(* Logix 5000 project; controller L3 vendor 1 type 14 code 92 rev 20.12; software revision 20.04; part 5 of 9 *)
(* tags used below, declared in another part *)
   B3 : DINT[100];
   cligno : BOOL;
   Status : INT;   // INT tag to retrieve Status value through GSV created during conversion
   T4 : TIMER[180];
   t_minute : TIMER;   // tempo on toutes les minute
   t_seconde : TIMER;   // tempo on toutes les secondes
   tcligno : TIMER;
(* _2_GENERAL, continued *)

ROUTINE _2_GENERAL   (* ladder *)
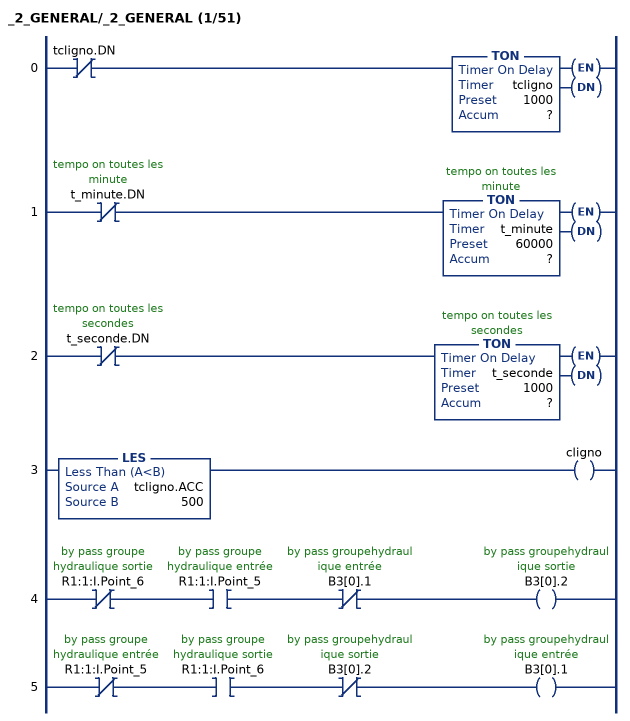
   0: XIO(tcligno.DN)TON(tcligno,?,?);
   1: XIO(t_minute.DN)TON(t_minute,?,?);
   2: XIO(t_seconde.DN)TON(t_seconde,?,?);
   3: LES(tcligno.ACC,500)OTE(cligno);
   4: XIO(R1:1:I.Point_6)XIC(R1:1:I.Point_5)XIO(B3[0].1)OTE(B3[0].2);
   5: XIO(R1:1:I.Point_5)XIC(R1:1:I.Point_6)XIO(B3[0].2)OTE(B3[0].1);
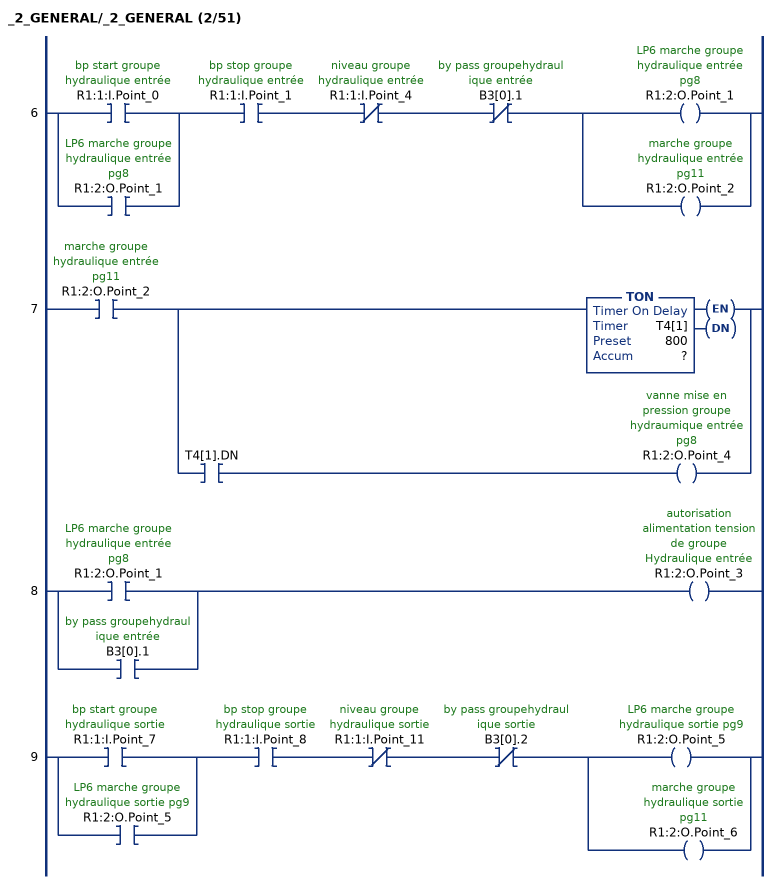
   6: [XIC(R1:1:I.Point_0) ,XIC(R1:2:O.Point_1) ]XIC(R1:1:I.Point_1)XIO(R1:1:I.Point_4)XIO(B3[0].1)[OTE(R1:2:O.Point_1) ,OTE(R1:2:O.Point_2) ];
   7: XIC(R1:2:O.Point_2)[TON(T4[1],?,?) ,XIC(T4[1].DN) OTE(R1:2:O.Point_4) ];
   8: [XIC(R1:2:O.Point_1) ,XIC(B3[0].1) ]OTE(R1:2:O.Point_3);
   9: [XIC(R1:1:I.Point_7) ,XIC(R1:2:O.Point_5) ]XIC(R1:1:I.Point_8)XIO(R1:1:I.Point_11)XIO(B3[0].2)[OTE(R1:2:O.Point_5) ,OTE(R1:2:O.Point_6) ];
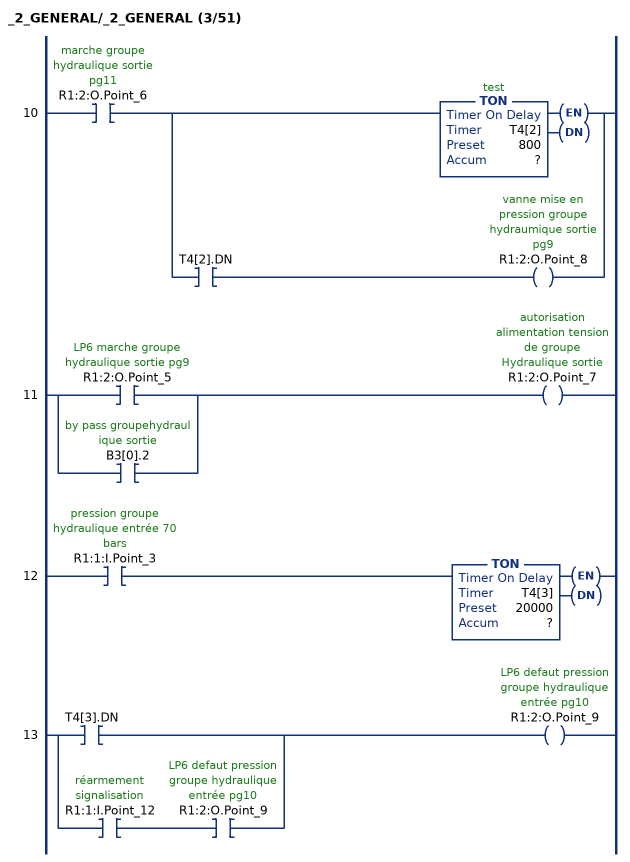
   10: XIC(R1:2:O.Point_6)[TON(T4[2],?,?) ,XIC(T4[2].DN) OTE(R1:2:O.Point_8) ];
   11: [XIC(R1:2:O.Point_5) ,XIC(B3[0].2) ]OTE(R1:2:O.Point_7);
   12: XIC(R1:1:I.Point_3)TON(T4[3],?,?);
   13: [XIC(T4[3].DN) ,XIC(R1:1:I.Point_12) XIC(R1:2:O.Point_9) ]OTE(R1:2:O.Point_9);
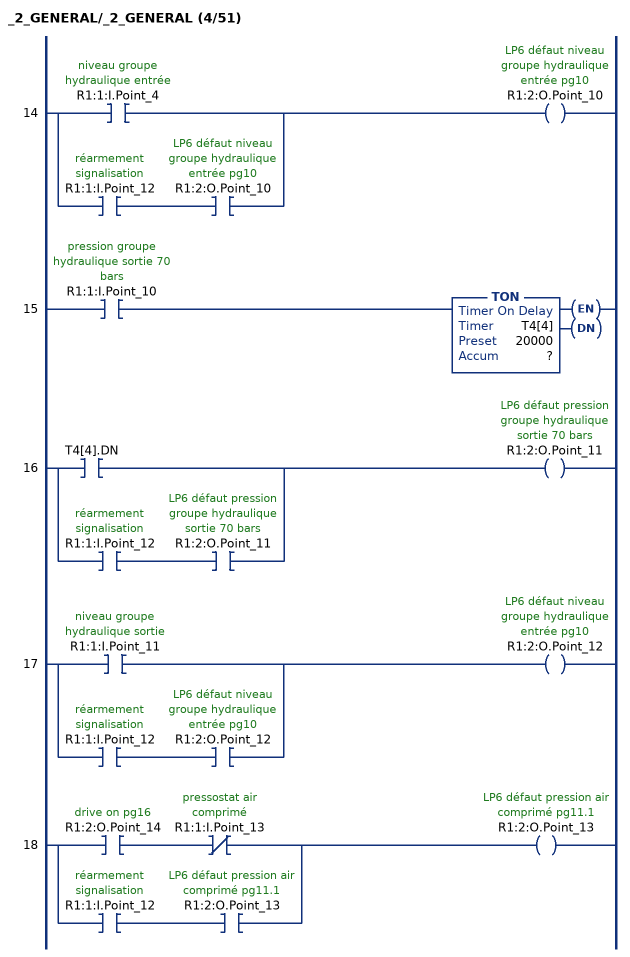
   14: [XIC(R1:1:I.Point_4) ,XIC(R1:1:I.Point_12) XIC(R1:2:O.Point_10) ]OTE(R1:2:O.Point_10);
   15: XIC(R1:1:I.Point_10)TON(T4[4],?,?);
   16: [XIC(T4[4].DN) ,XIC(R1:1:I.Point_12) XIC(R1:2:O.Point_11) ]OTE(R1:2:O.Point_11);
   17: [XIC(R1:1:I.Point_11) ,XIC(R1:1:I.Point_12) XIC(R1:2:O.Point_12) ]OTE(R1:2:O.Point_12);
   18: [XIC(R1:2:O.Point_14) XIO(R1:1:I.Point_13) ,XIC(R1:1:I.Point_12) XIC(R1:2:O.Point_13) ]OTE(R1:2:O.Point_13);
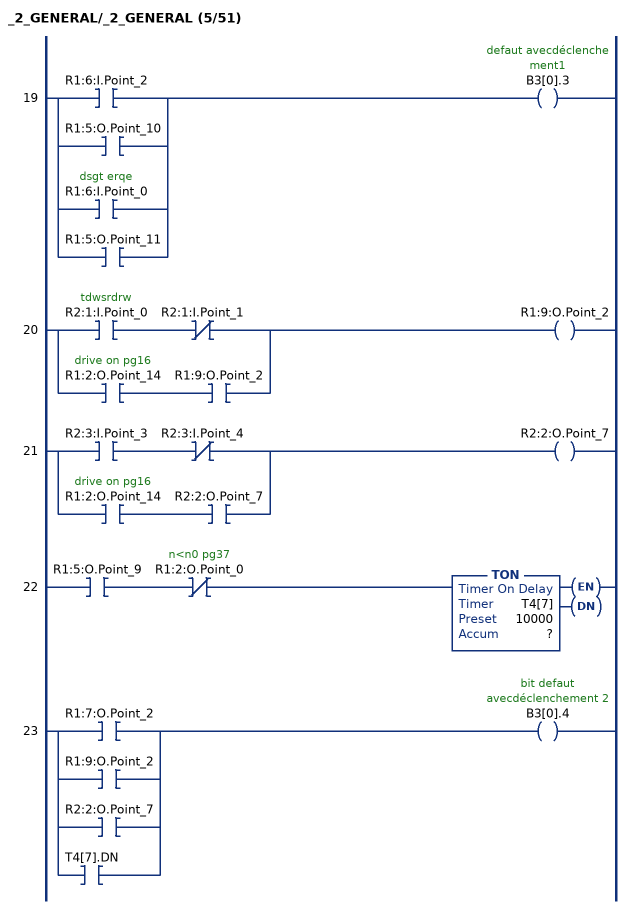
   19: [XIC(R1:6:I.Point_2) ,XIC(R1:5:O.Point_10) ,XIC(R1:6:I.Point_0) ,XIC(R1:5:O.Point_11) ]OTE(B3[0].3);
   20: [XIC(R2:1:I.Point_0) XIO(R2:1:I.Point_1) ,XIC(R1:2:O.Point_14) XIC(R1:9:O.Point_2) ]OTE(R1:9:O.Point_2);
   21: [XIC(R2:3:I.Point_3) XIO(R2:3:I.Point_4) ,XIC(R1:2:O.Point_14) XIC(R2:2:O.Point_7) ]OTE(R2:2:O.Point_7);
   22: XIC(R1:5:O.Point_9)XIO(R1:2:O.Point_0)TON(T4[7],?,?);
   23: [XIC(R1:7:O.Point_2) ,XIC(R1:9:O.Point_2) ,XIC(R2:2:O.Point_7) ,XIC(T4[7].DN) ]OTE(B3[0].4);
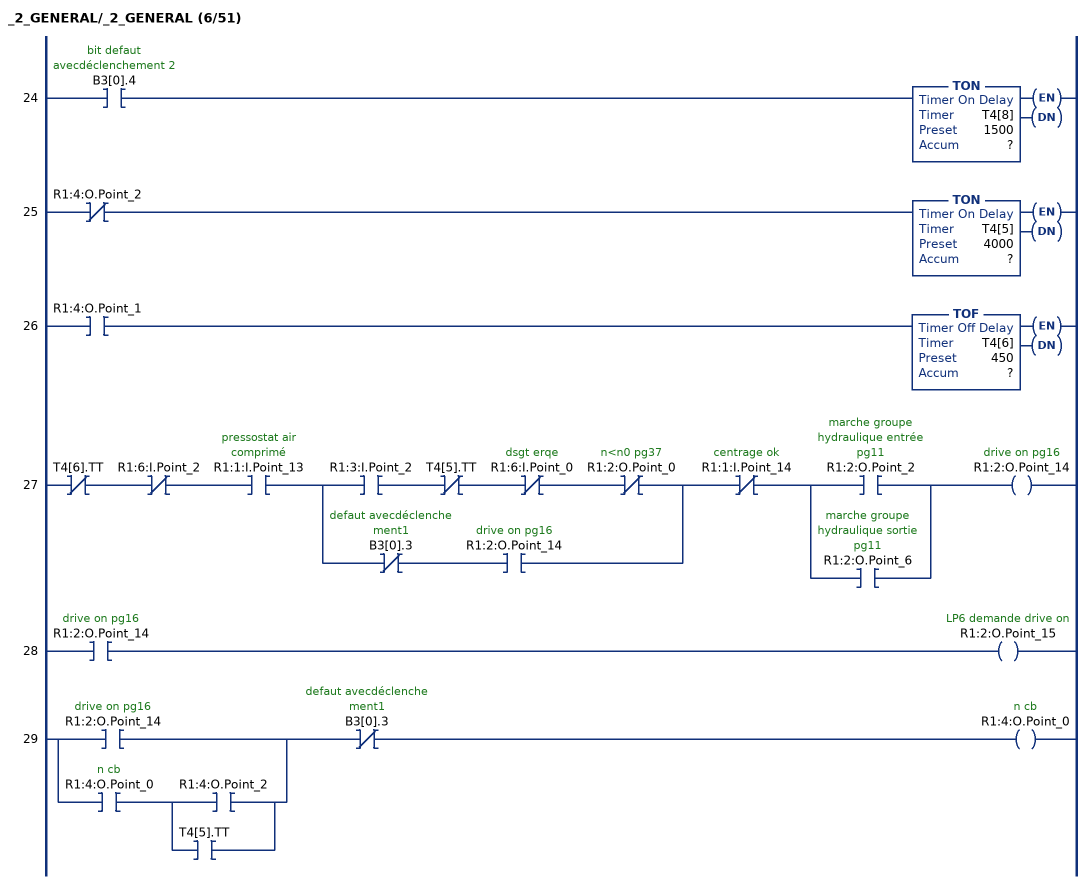
   24: XIC(B3[0].4)TON(T4[8],?,?);
   25: XIO(R1:4:O.Point_2)TON(T4[5],?,?);
   26: XIC(R1:4:O.Point_1)TOF(T4[6],?,?);
   27: XIO(T4[6].TT)XIO(R1:6:I.Point_2)XIC(R1:1:I.Point_13)[XIC(R1:3:I.Point_2) XIO(T4[5].TT) XIO(R1:6:I.Point_0) XIO(R1:2:O.Point_0) ,XIO(B3[0].3) XIC(R1:2:O.Point_14) ]XIO(R1:1:I.Point_14)[XIC(R1:2:O.Point_2) ,XIC(R1:2:O.Point_6) ]OTE(R1:2:O.Point_14);
   28: XIC(R1:2:O.Point_14)OTE(R1:2:O.Point_15);
   29: [XIC(R1:2:O.Point_14) ,XIC(R1:4:O.Point_0) [XIC(R1:4:O.Point_2) ,XIC(T4[5].TT) ] ]XIO(B3[0].3)OTE(R1:4:O.Point_0);
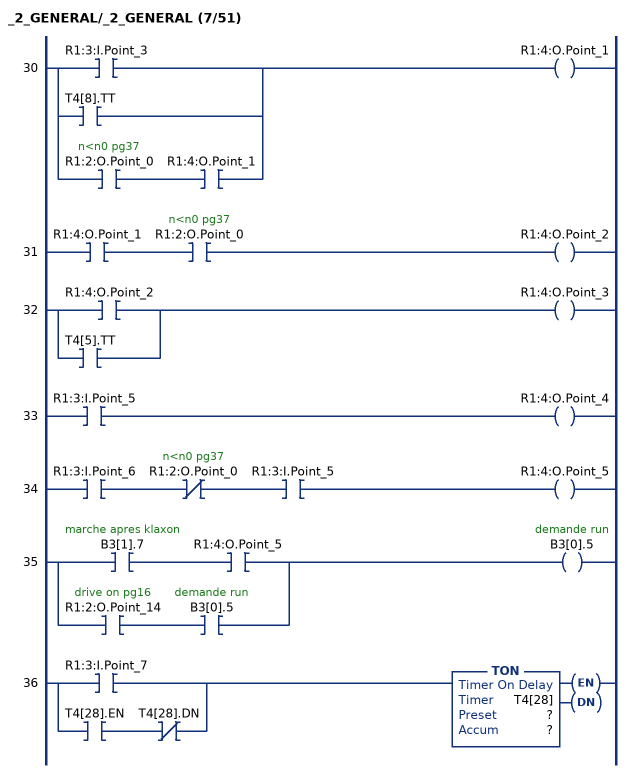
   30: [XIC(R1:3:I.Point_3) ,XIC(T4[8].TT) ,XIC(R1:2:O.Point_0) XIC(R1:4:O.Point_1) ]OTE(R1:4:O.Point_1);
   31: XIC(R1:4:O.Point_1)XIC(R1:2:O.Point_0)OTE(R1:4:O.Point_2);
   32: [XIC(R1:4:O.Point_2) ,XIC(T4[5].TT) ]OTE(R1:4:O.Point_3);
   33: XIC(R1:3:I.Point_5)OTE(R1:4:O.Point_4);
   34: XIC(R1:3:I.Point_6)XIO(R1:2:O.Point_0)XIC(R1:3:I.Point_5)OTE(R1:4:O.Point_5);
   35: [XIC(B3[1].7) XIC(R1:4:O.Point_5) ,XIC(R1:2:O.Point_14) XIC(B3[0].5) ]OTE(B3[0].5);
   36: [XIC(R1:3:I.Point_7) ,XIC(T4[28].EN) XIO(T4[28].DN) ]TON(T4[28],?,?);
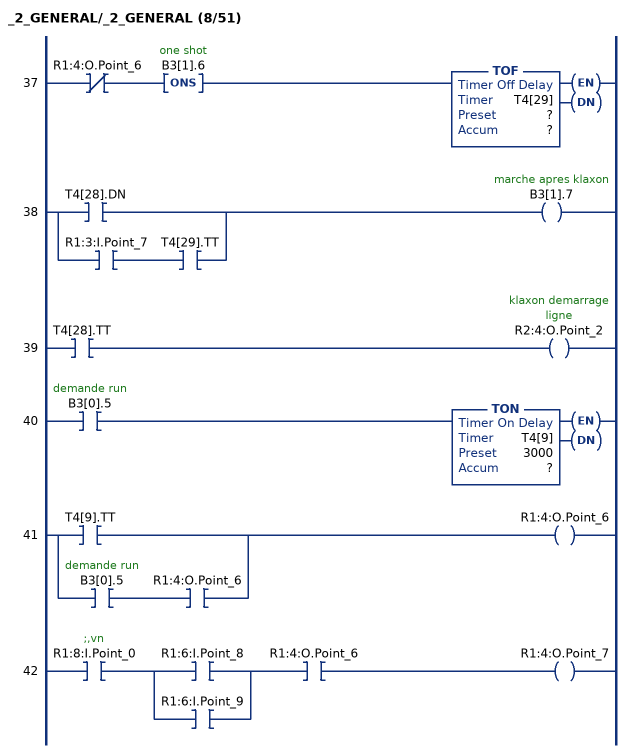
   37: XIO(R1:4:O.Point_6)ONS(B3[1].6)TOF(T4[29],?,?);
   38: [XIC(T4[28].DN) ,XIC(R1:3:I.Point_7) XIC(T4[29].TT) ]OTE(B3[1].7);
   39: XIC(T4[28].TT)OTE(R2:4:O.Point_2);
   40: XIC(B3[0].5)TON(T4[9],?,?);
   41: [XIC(T4[9].TT) ,XIC(B3[0].5) XIC(R1:4:O.Point_6) ]OTE(R1:4:O.Point_6);
   42: XIC(R1:8:I.Point_0)[XIC(R1:6:I.Point_8) ,XIC(R1:6:I.Point_9) ]XIC(R1:4:O.Point_6)OTE(R1:4:O.Point_7);
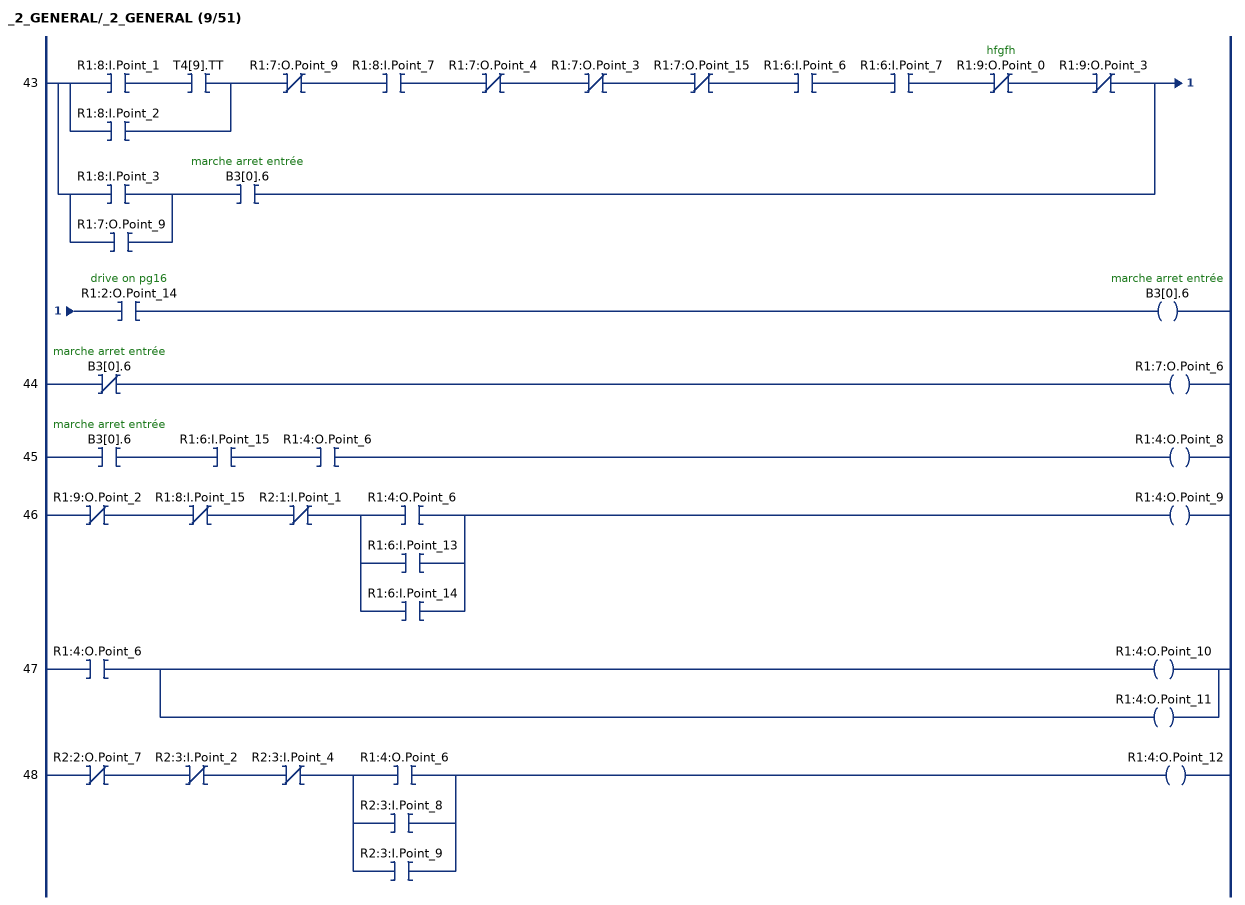
   43: [[XIC(R1:8:I.Point_1) XIC(T4[9].TT) ,XIC(R1:8:I.Point_2) ] XIO(R1:7:O.Point_9) XIC(R1:8:I.Point_7) XIO(R1:7:O.Point_4) XIO(R1:7:O.Point_3) XIO(R1:7:O.Point_15) XIC(R1:6:I.Point_6) XIC(R1:6:I.Point_7) XIO(R1:9:O.Point_0) XIO(R1:9:O.Point_3) ,[XIC(R1:8:I.Point_3) ,XIC(R1:7:O.Point_9) ] XIC(B3[0].6) ]XIC(R1:2:O.Point_14)OTE(B3[0].6);
   44: XIO(B3[0].6)OTE(R1:7:O.Point_6);
   45: XIC(B3[0].6)XIC(R1:6:I.Point_15)XIC(R1:4:O.Point_6)OTE(R1:4:O.Point_8);
   46: XIO(R1:9:O.Point_2)XIO(R1:8:I.Point_15)XIO(R2:1:I.Point_1)[XIC(R1:4:O.Point_6) ,XIC(R1:6:I.Point_13) ,XIC(R1:6:I.Point_14) ]OTE(R1:4:O.Point_9);
   47: XIC(R1:4:O.Point_6)[OTE(R1:4:O.Point_10) ,OTE(R1:4:O.Point_11) ];
   48: XIO(R2:2:O.Point_7)XIO(R2:3:I.Point_2)XIO(R2:3:I.Point_4)[XIC(R1:4:O.Point_6) ,XIC(R2:3:I.Point_8) ,XIC(R2:3:I.Point_9) ]OTE(R1:4:O.Point_12);
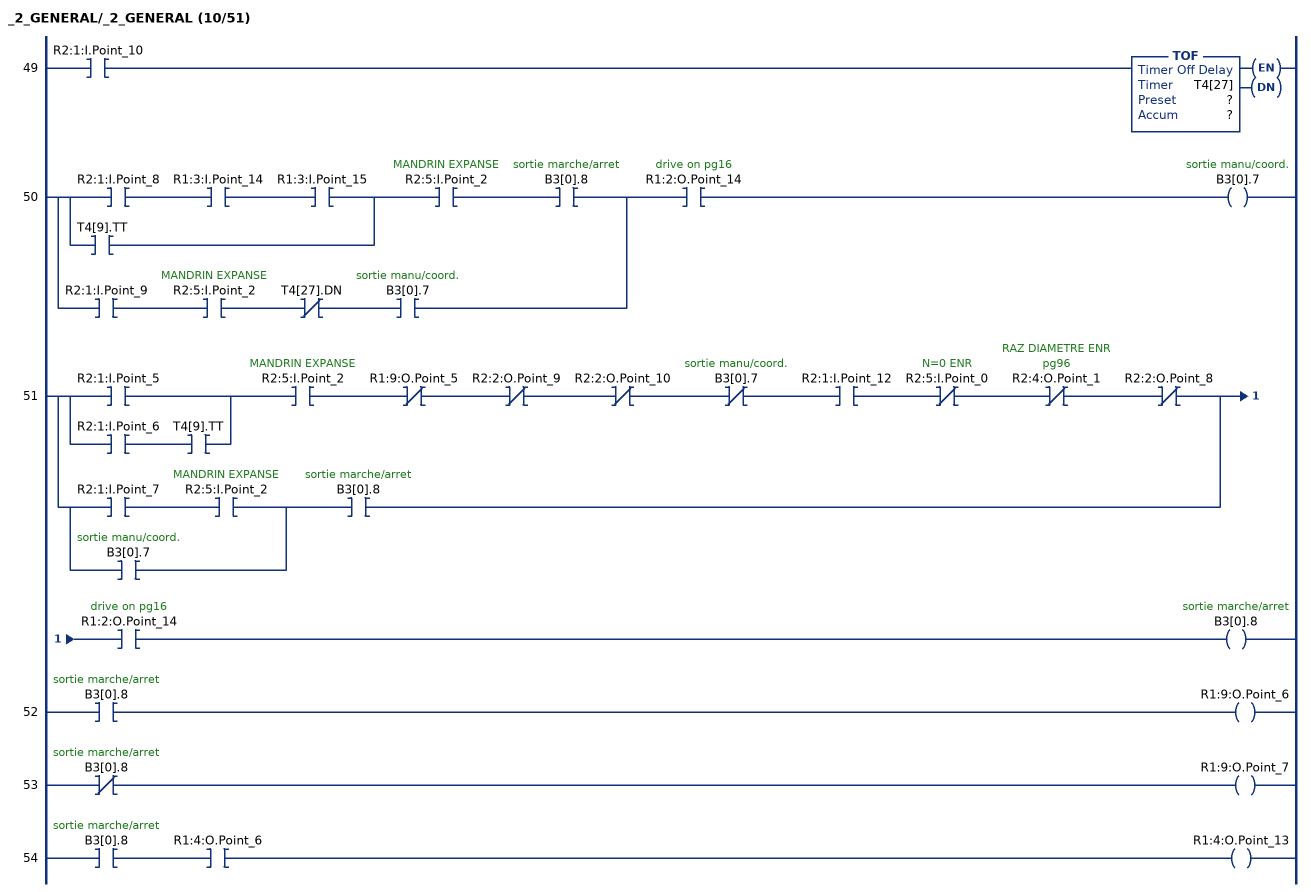
   49: XIC(R2:1:I.Point_10)TOF(T4[27],?,?);
   50: [[XIC(R2:1:I.Point_8) XIC(R1:3:I.Point_14) XIC(R1:3:I.Point_15) ,XIC(T4[9].TT) ] XIC(R2:5:I.Point_2) XIC(B3[0].8) ,XIC(R2:1:I.Point_9) XIC(R2:5:I.Point_2) XIO(T4[27].DN) XIC(B3[0].7) ]XIC(R1:2:O.Point_14)OTE(B3[0].7);
   51: [[XIC(R2:1:I.Point_5) ,XIC(R2:1:I.Point_6) XIC(T4[9].TT) ] XIC(R2:5:I.Point_2) XIO(R1:9:O.Point_5) XIO(R2:2:O.Point_9) XIO(R2:2:O.Point_10) XIO(B3[0].7) XIC(R2:1:I.Point_12) XIO(R2:5:I.Point_0) XIO(R2:4:O.Point_1) XIO(R2:2:O.Point_8) ,[XIC(R2:1:I.Point_7) XIC(R2:5:I.Point_2) ,XIC(B3[0].7) ] XIC(B3[0].8) ]XIC(R1:2:O.Point_14)OTE(B3[0].8);
   52: XIC(B3[0].8)OTE(R1:9:O.Point_6);
   53: XIO(B3[0].8)OTE(R1:9:O.Point_7);
   54: XIC(B3[0].8)XIC(R1:4:O.Point_6)OTE(R1:4:O.Point_13);
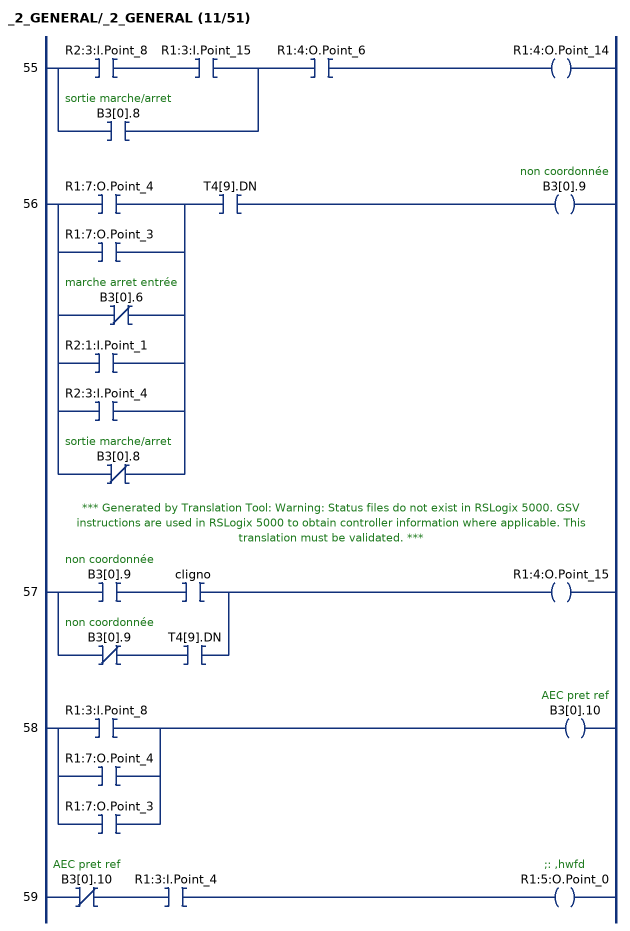
   55: [XIC(R2:3:I.Point_8) XIC(R1:3:I.Point_15) ,XIC(B3[0].8) ]XIC(R1:4:O.Point_6)OTE(R1:4:O.Point_14);
   56: [XIC(R1:7:O.Point_4) ,XIC(R1:7:O.Point_3) ,XIO(B3[0].6) ,XIC(R2:1:I.Point_1) ,XIC(R2:3:I.Point_4) ,XIO(B3[0].8) ]XIC(T4[9].DN)OTE(B3[0].9);
   // *** Generated by Translation Tool: Warning: Status files do not exist in RSLogix 5000. GSV instructions are used in RSLogix 5000 to obtain controller information where applicable. This translation must be validated. ***
   57: [XIC(B3[0].9) XIC(cligno) ,XIO(B3[0].9) XIC(T4[9].DN) ]OTE(R1:4:O.Point_15);
   58: [XIC(R1:3:I.Point_8) ,XIC(R1:7:O.Point_4) ,XIC(R1:7:O.Point_3) ]OTE(B3[0].10);
   59: XIO(B3[0].10)XIC(R1:3:I.Point_4)OTE(R1:5:O.Point_0);
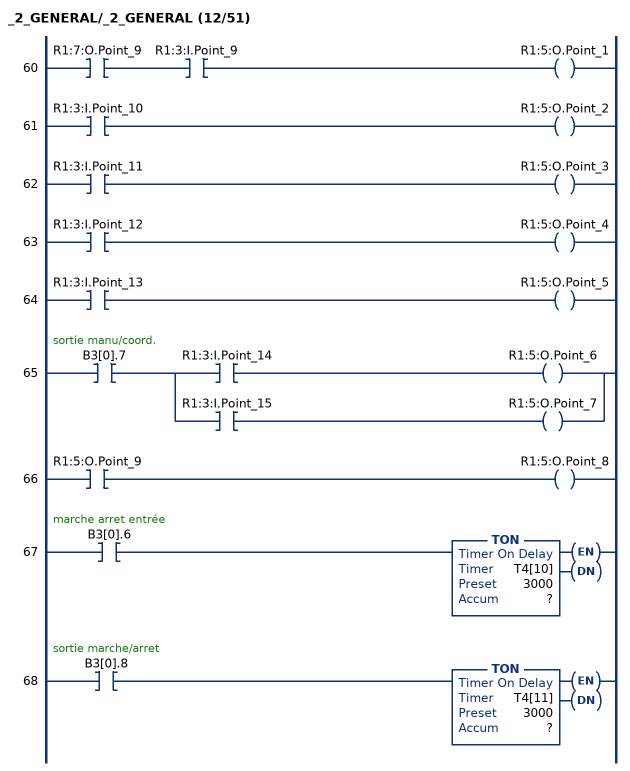
   60: XIC(R1:7:O.Point_9)XIC(R1:3:I.Point_9)OTE(R1:5:O.Point_1);
   61: XIC(R1:3:I.Point_10)OTE(R1:5:O.Point_2);
   62: XIC(R1:3:I.Point_11)OTE(R1:5:O.Point_3);
   63: XIC(R1:3:I.Point_12)OTE(R1:5:O.Point_4);
   64: XIC(R1:3:I.Point_13)OTE(R1:5:O.Point_5);
   65: XIC(B3[0].7)[XIC(R1:3:I.Point_14) OTE(R1:5:O.Point_6) ,XIC(R1:3:I.Point_15) OTE(R1:5:O.Point_7) ];
   66: XIC(R1:5:O.Point_9)OTE(R1:5:O.Point_8);
   67: XIC(B3[0].6)TON(T4[10],?,?);
   68: XIC(B3[0].8)TON(T4[11],?,?);
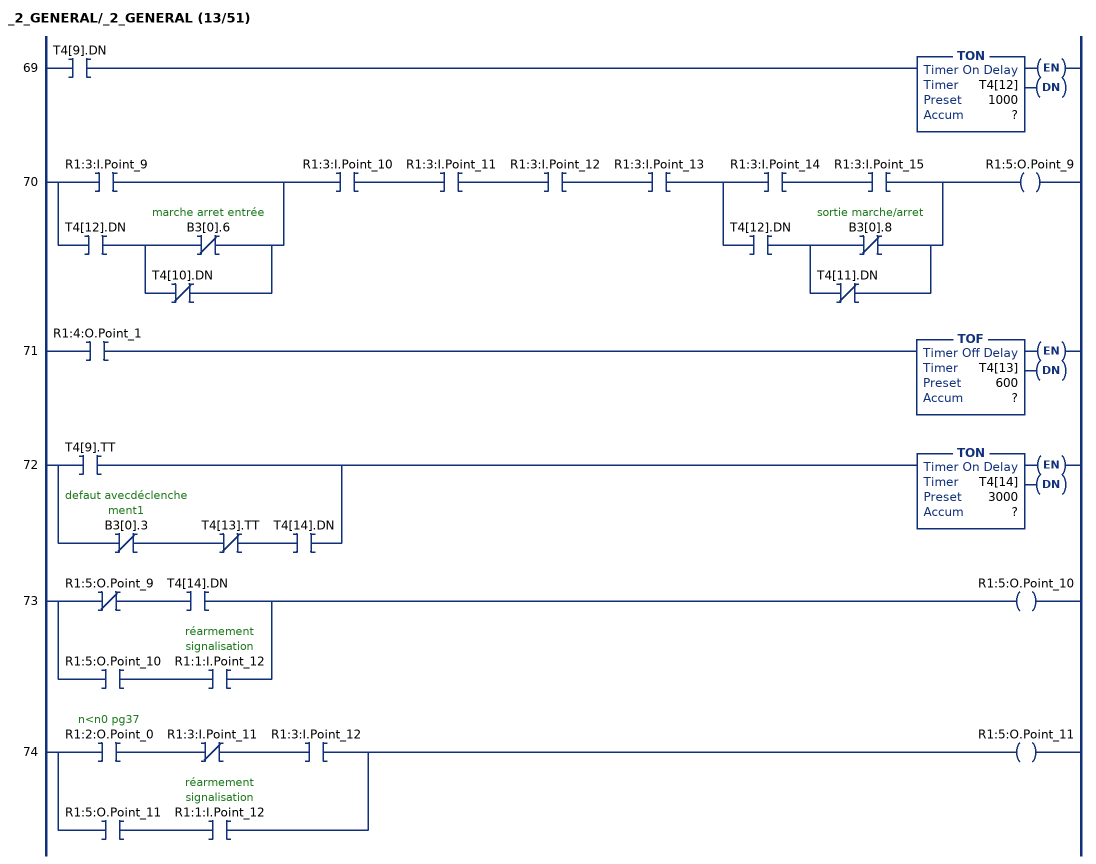
   69: XIC(T4[9].DN)TON(T4[12],?,?);
   70: [XIC(R1:3:I.Point_9) ,XIC(T4[12].DN) [XIO(B3[0].6) ,XIO(T4[10].DN) ] ]XIC(R1:3:I.Point_10)XIC(R1:3:I.Point_11)XIC(R1:3:I.Point_12)XIC(R1:3:I.Point_13)[XIC(R1:3:I.Point_14) XIC(R1:3:I.Point_15) ,XIC(T4[12].DN) [XIO(B3[0].8) ,XIO(T4[11].DN) ] ]OTE(R1:5:O.Point_9);
   71: XIC(R1:4:O.Point_1)TOF(T4[13],?,?);
   72: [XIC(T4[9].TT) ,XIO(B3[0].3) XIO(T4[13].TT) XIC(T4[14].DN) ]TON(T4[14],?,?);
   73: [XIO(R1:5:O.Point_9) XIC(T4[14].DN) ,XIC(R1:5:O.Point_10) XIC(R1:1:I.Point_12) ]OTE(R1:5:O.Point_10);
   74: [XIC(R1:2:O.Point_0) XIO(R1:3:I.Point_11) XIC(R1:3:I.Point_12) ,XIC(R1:5:O.Point_11) XIC(R1:1:I.Point_12) ]OTE(R1:5:O.Point_11);
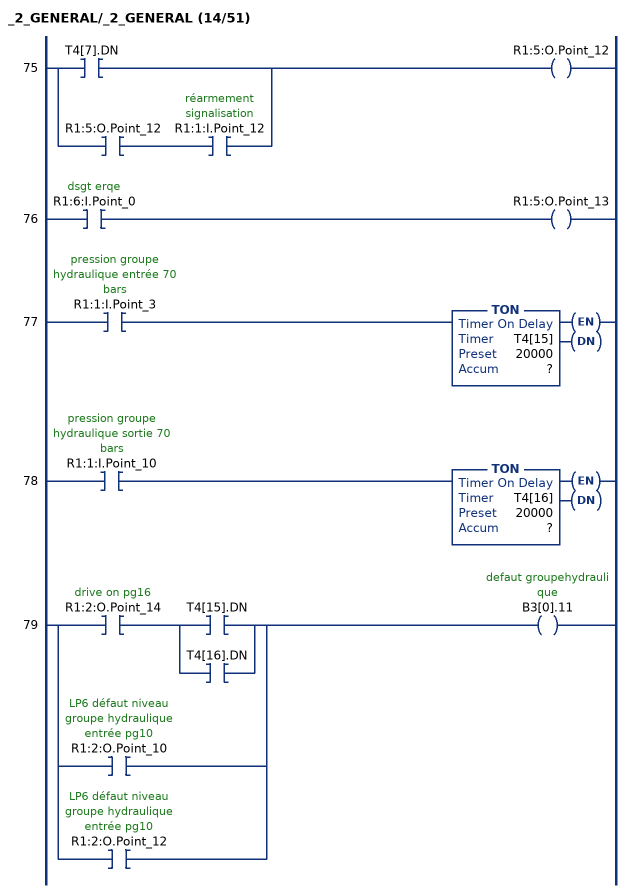
   75: [XIC(T4[7].DN) ,XIC(R1:5:O.Point_12) XIC(R1:1:I.Point_12) ]OTE(R1:5:O.Point_12);
   76: XIC(R1:6:I.Point_0)OTE(R1:5:O.Point_13);
   77: XIC(R1:1:I.Point_3)TON(T4[15],?,?);
   78: XIC(R1:1:I.Point_10)TON(T4[16],?,?);
   79: [XIC(R1:2:O.Point_14) [XIC(T4[15].DN) ,XIC(T4[16].DN) ] ,XIC(R1:2:O.Point_10) ,XIC(R1:2:O.Point_12) ]OTE(B3[0].11);
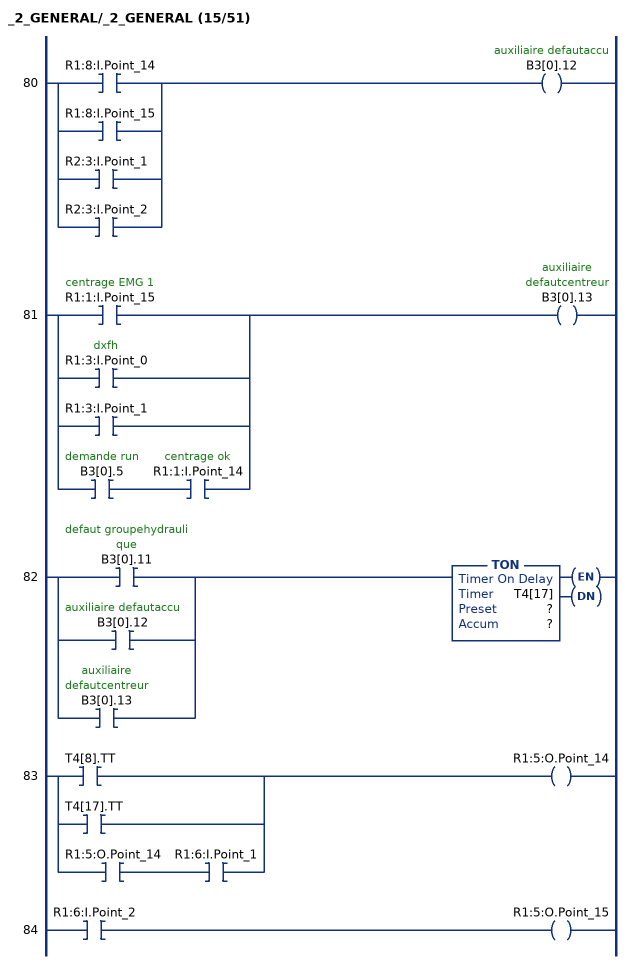
   80: [XIC(R1:8:I.Point_14) ,XIC(R1:8:I.Point_15) ,XIC(R2:3:I.Point_1) ,XIC(R2:3:I.Point_2) ]OTE(B3[0].12);
   81: [XIC(R1:1:I.Point_15) ,XIC(R1:3:I.Point_0) ,XIC(R1:3:I.Point_1) ,XIC(B3[0].5) XIC(R1:1:I.Point_14) ]OTE(B3[0].13);
   82: [XIC(B3[0].11) ,XIC(B3[0].12) ,XIC(B3[0].13) ]TON(T4[17],?,?);
   83: [XIC(T4[8].TT) ,XIC(T4[17].TT) ,XIC(R1:5:O.Point_14) XIC(R1:6:I.Point_1) ]OTE(R1:5:O.Point_14);
   84: XIC(R1:6:I.Point_2)OTE(R1:5:O.Point_15);
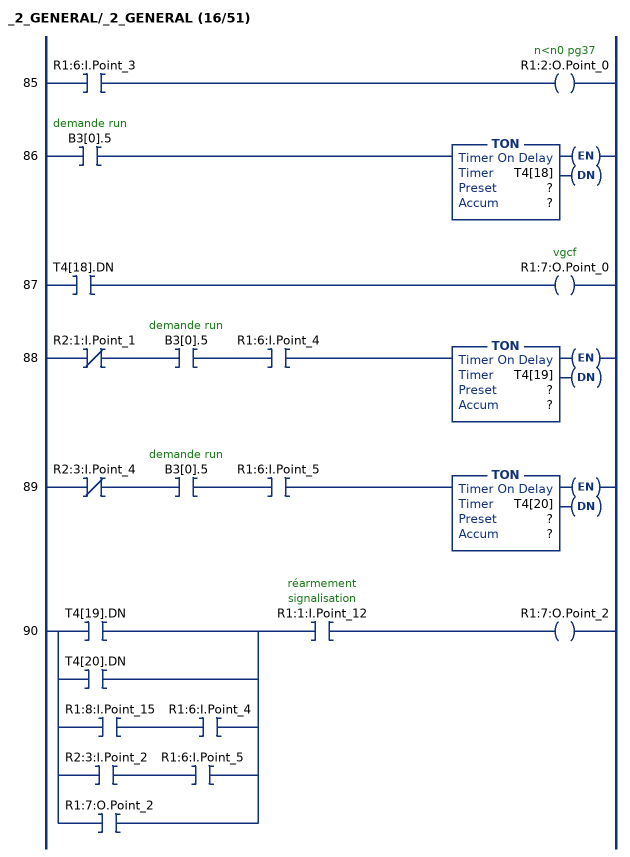
   85: XIC(R1:6:I.Point_3)OTE(R1:2:O.Point_0);
   86: XIC(B3[0].5)TON(T4[18],?,?);
   87: XIC(T4[18].DN)OTE(R1:7:O.Point_0);
   88: XIO(R2:1:I.Point_1)XIC(B3[0].5)XIC(R1:6:I.Point_4)TON(T4[19],?,?);
   89: XIO(R2:3:I.Point_4)XIC(B3[0].5)XIC(R1:6:I.Point_5)TON(T4[20],?,?);
   90: [XIC(T4[19].DN) ,XIC(T4[20].DN) ,XIC(R1:8:I.Point_15) XIC(R1:6:I.Point_4) ,XIC(R2:3:I.Point_2) XIC(R1:6:I.Point_5) ,XIC(R1:7:O.Point_2) ]XIC(R1:1:I.Point_12)OTE(R1:7:O.Point_2);
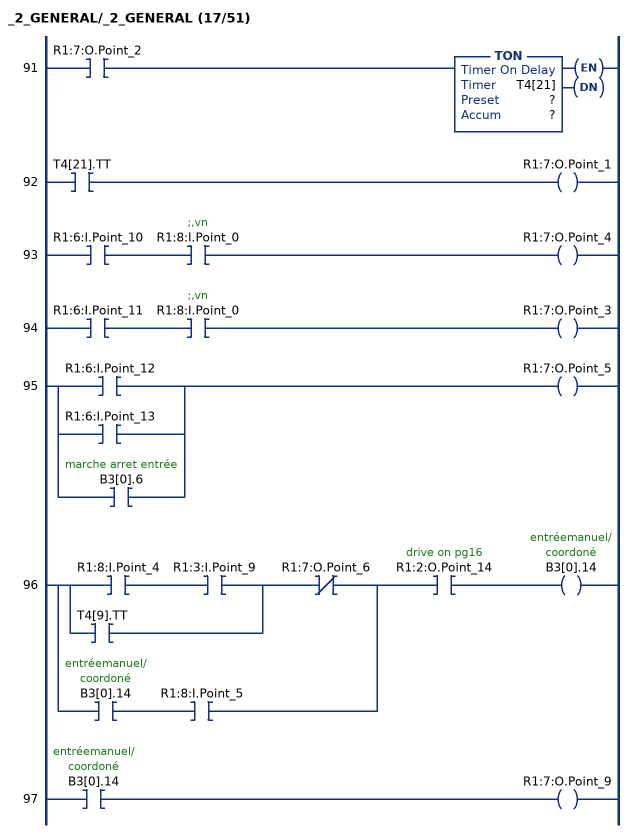
   91: XIC(R1:7:O.Point_2)TON(T4[21],?,?);
   92: XIC(T4[21].TT)OTE(R1:7:O.Point_1);
   93: XIC(R1:6:I.Point_10)XIC(R1:8:I.Point_0)OTE(R1:7:O.Point_4);
   94: XIC(R1:6:I.Point_11)XIC(R1:8:I.Point_0)OTE(R1:7:O.Point_3);
   95: [XIC(R1:6:I.Point_12) ,XIC(R1:6:I.Point_13) ,XIC(B3[0].6) ]OTE(R1:7:O.Point_5);
   96: [[XIC(R1:8:I.Point_4) XIC(R1:3:I.Point_9) ,XIC(T4[9].TT) ] XIO(R1:7:O.Point_6) ,XIC(B3[0].14) XIC(R1:8:I.Point_5) ]XIC(R1:2:O.Point_14)OTE(B3[0].14);
   97: XIC(B3[0].14)OTE(R1:7:O.Point_9);
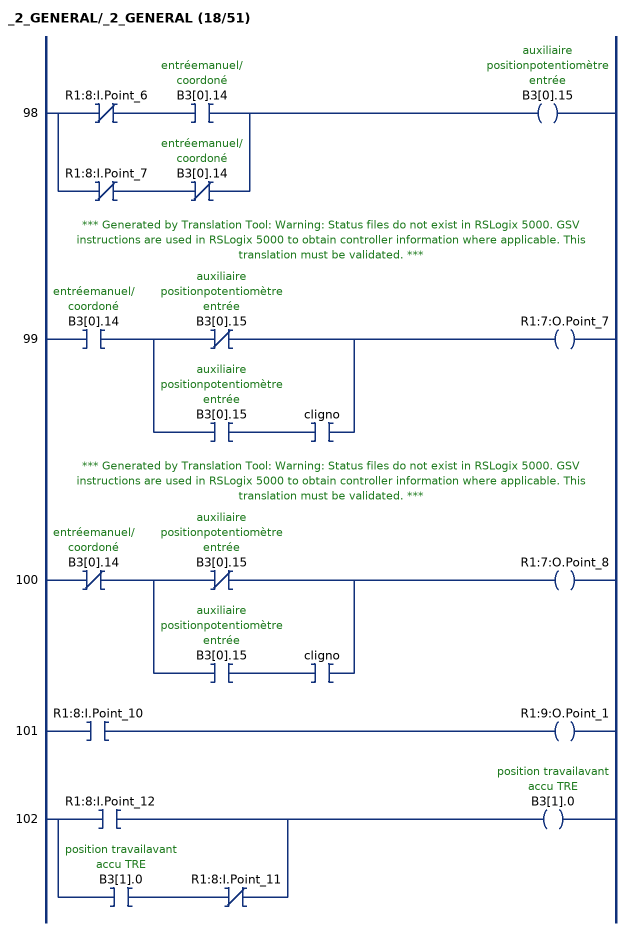
   98: [XIO(R1:8:I.Point_6) XIC(B3[0].14) ,XIO(R1:8:I.Point_7) XIO(B3[0].14) ]OTE(B3[0].15);
   // *** Generated by Translation Tool: Warning: Status files do not exist in RSLogix 5000. GSV instructions are used in RSLogix 5000 to obtain controller information where applicable. This translation must be validated. ***
   99: XIC(B3[0].14)[XIO(B3[0].15) ,XIC(B3[0].15) XIC(cligno) ]OTE(R1:7:O.Point_7);
   // *** Generated by Translation Tool: Warning: Status files do not exist in RSLogix 5000. GSV instructions are used in RSLogix 5000 to obtain controller information where applicable. This translation must be validated. ***
   100: XIO(B3[0].14)[XIO(B3[0].15) ,XIC(B3[0].15) XIC(cligno) ]OTE(R1:7:O.Point_8);
   101: XIC(R1:8:I.Point_10)OTE(R1:9:O.Point_1);
   102: [XIC(R1:8:I.Point_12) ,XIC(B3[1].0) XIO(R1:8:I.Point_11) ]OTE(B3[1].0);
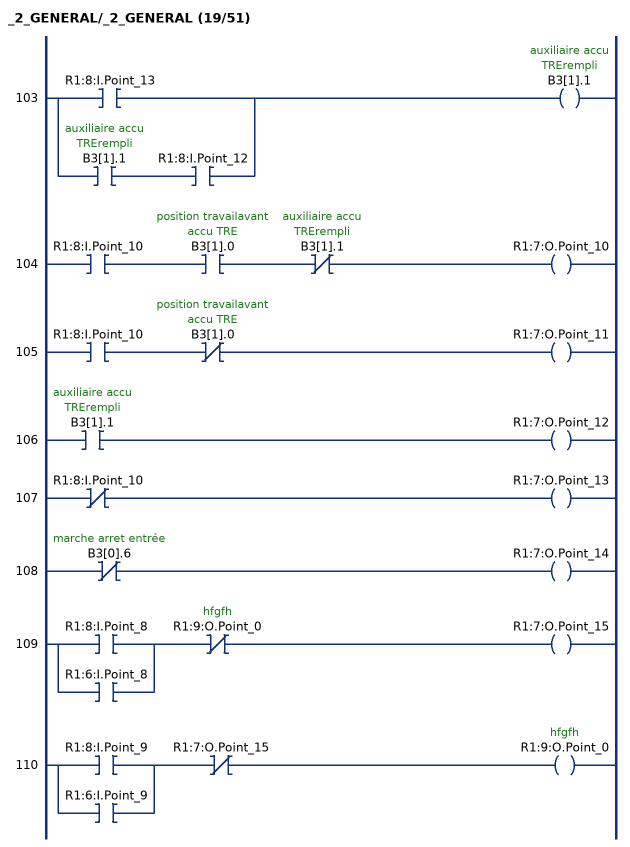
   103: [XIC(R1:8:I.Point_13) ,XIC(B3[1].1) XIC(R1:8:I.Point_12) ]OTE(B3[1].1);
   104: XIC(R1:8:I.Point_10)XIC(B3[1].0)XIO(B3[1].1)OTE(R1:7:O.Point_10);
   105: XIC(R1:8:I.Point_10)XIO(B3[1].0)OTE(R1:7:O.Point_11);
   106: XIC(B3[1].1)OTE(R1:7:O.Point_12);
   107: XIO(R1:8:I.Point_10)OTE(R1:7:O.Point_13);
   108: XIO(B3[0].6)OTE(R1:7:O.Point_14);
   109: [XIC(R1:8:I.Point_8) ,XIC(R1:6:I.Point_8) ]XIO(R1:9:O.Point_0)OTE(R1:7:O.Point_15);
   110: [XIC(R1:8:I.Point_9) ,XIC(R1:6:I.Point_9) ]XIO(R1:7:O.Point_15)OTE(R1:9:O.Point_0);
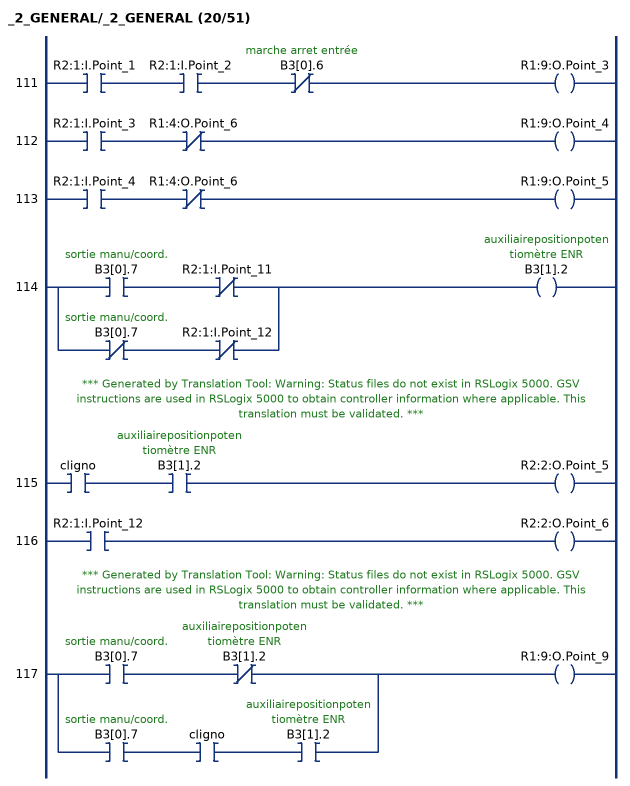
   111: XIC(R2:1:I.Point_1)XIC(R2:1:I.Point_2)XIO(B3[0].6)OTE(R1:9:O.Point_3);
   112: XIC(R2:1:I.Point_3)XIO(R1:4:O.Point_6)OTE(R1:9:O.Point_4);
   113: XIC(R2:1:I.Point_4)XIO(R1:4:O.Point_6)OTE(R1:9:O.Point_5);
   114: [XIC(B3[0].7) XIO(R2:1:I.Point_11) ,XIO(B3[0].7) XIO(R2:1:I.Point_12) ]OTE(B3[1].2);
   // *** Generated by Translation Tool: Warning: Status files do not exist in RSLogix 5000. GSV instructions are used in RSLogix 5000 to obtain controller information where applicable. This translation must be validated. ***
   115: XIC(cligno)XIC(B3[1].2)OTE(R2:2:O.Point_5);
   116: XIC(R2:1:I.Point_12)OTE(R2:2:O.Point_6);
   // *** Generated by Translation Tool: Warning: Status files do not exist in RSLogix 5000. GSV instructions are used in RSLogix 5000 to obtain controller information where applicable. This translation must be validated. ***
   117: [XIC(B3[0].7) XIO(B3[1].2) ,XIC(B3[0].7) XIC(cligno) XIC(B3[1].2) ]OTE(R1:9:O.Point_9);
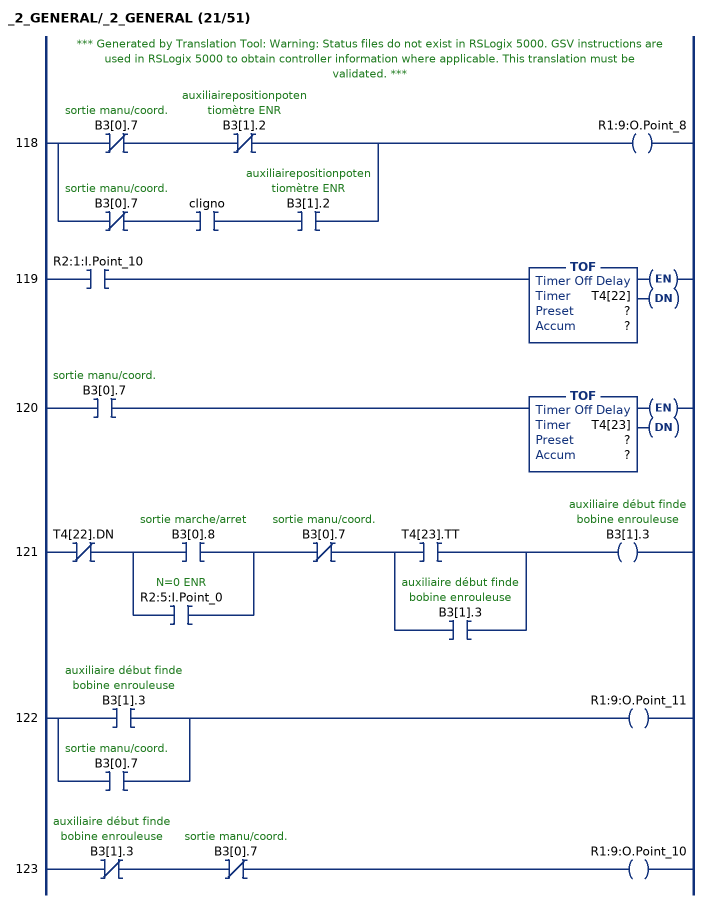
   // *** Generated by Translation Tool: Warning: Status files do not exist in RSLogix 5000. GSV instructions are used in RSLogix 5000 to obtain controller information where applicable. This translation must be validated. ***
   118: [XIO(B3[0].7) XIO(B3[1].2) ,XIO(B3[0].7) XIC(cligno) XIC(B3[1].2) ]OTE(R1:9:O.Point_8);
   119: XIC(R2:1:I.Point_10)TOF(T4[22],?,?);
   120: XIC(B3[0].7)TOF(T4[23],?,?);
   121: XIO(T4[22].DN)[XIC(B3[0].8) ,XIC(R2:5:I.Point_0) ]XIO(B3[0].7)[XIC(T4[23].TT) ,XIC(B3[1].3) ]OTE(B3[1].3);
   122: [XIC(B3[1].3) ,XIC(B3[0].7) ]OTE(R1:9:O.Point_11);
   123: XIO(B3[1].3)XIO(B3[0].7)OTE(R1:9:O.Point_10);
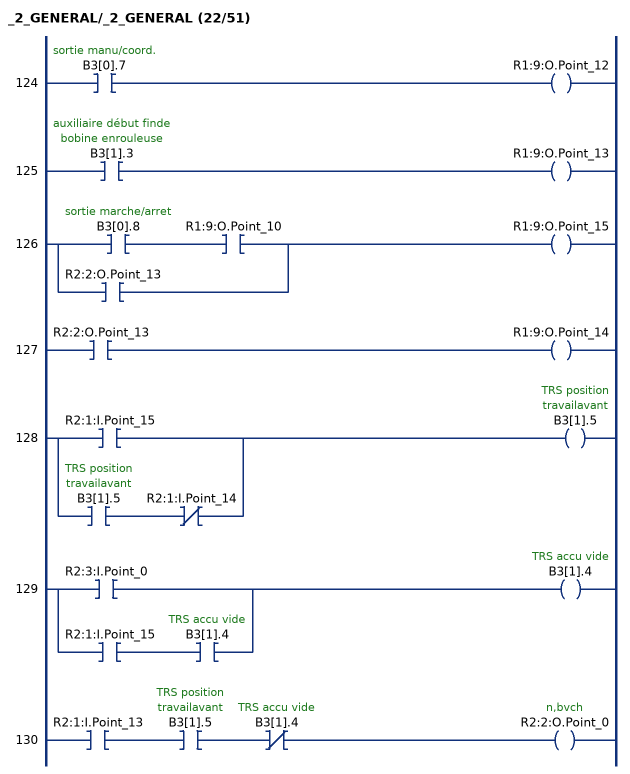
   124: XIC(B3[0].7)OTE(R1:9:O.Point_12);
   125: XIC(B3[1].3)OTE(R1:9:O.Point_13);
   126: [XIC(B3[0].8) XIC(R1:9:O.Point_10) ,XIC(R2:2:O.Point_13) ]OTE(R1:9:O.Point_15);
   127: XIC(R2:2:O.Point_13)OTE(R1:9:O.Point_14);
   128: [XIC(R2:1:I.Point_15) ,XIC(B3[1].5) XIO(R2:1:I.Point_14) ]OTE(B3[1].5);
   129: [XIC(R2:3:I.Point_0) ,XIC(R2:1:I.Point_15) XIC(B3[1].4) ]OTE(B3[1].4);
   130: XIC(R2:1:I.Point_13)XIC(B3[1].5)XIO(B3[1].4)OTE(R2:2:O.Point_0);
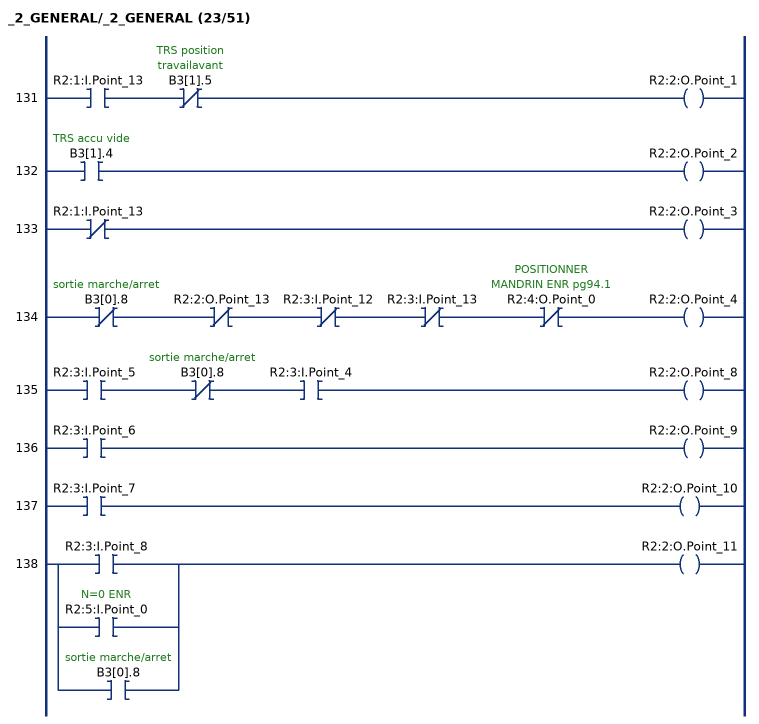
   131: XIC(R2:1:I.Point_13)XIO(B3[1].5)OTE(R2:2:O.Point_1);
   132: XIC(B3[1].4)OTE(R2:2:O.Point_2);
   133: XIO(R2:1:I.Point_13)OTE(R2:2:O.Point_3);
   134: XIO(B3[0].8)XIO(R2:2:O.Point_13)XIO(R2:3:I.Point_12)XIO(R2:3:I.Point_13)XIO(R2:4:O.Point_0)OTE(R2:2:O.Point_4);
   135: XIC(R2:3:I.Point_5)XIO(B3[0].8)XIC(R2:3:I.Point_4)OTE(R2:2:O.Point_8);
   136: XIC(R2:3:I.Point_6)OTE(R2:2:O.Point_9);
   137: XIC(R2:3:I.Point_7)OTE(R2:2:O.Point_10);
   138: [XIC(R2:3:I.Point_8) ,XIC(R2:5:I.Point_0) ,XIC(B3[0].8) ]OTE(R2:2:O.Point_11);
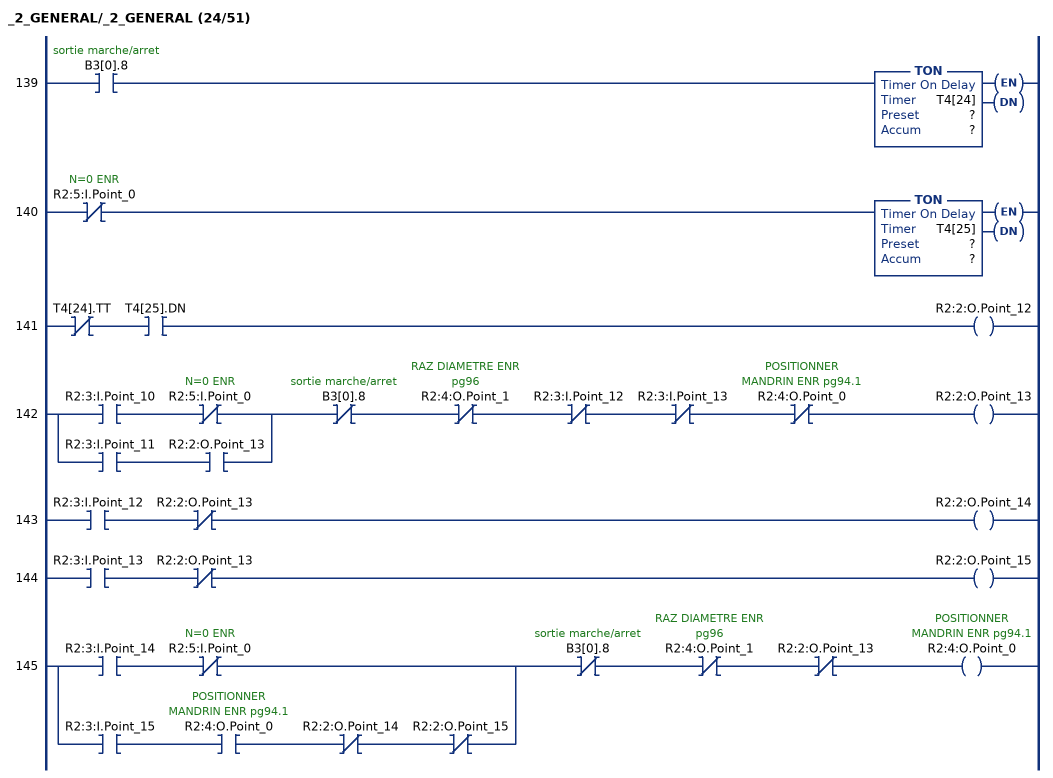
   139: XIC(B3[0].8)TON(T4[24],?,?);
   140: XIO(R2:5:I.Point_0)TON(T4[25],?,?);
   141: XIO(T4[24].TT)XIC(T4[25].DN)OTE(R2:2:O.Point_12);
   142: [XIC(R2:3:I.Point_10) XIO(R2:5:I.Point_0) ,XIC(R2:3:I.Point_11) XIC(R2:2:O.Point_13) ]XIO(B3[0].8)XIO(R2:4:O.Point_1)XIO(R2:3:I.Point_12)XIO(R2:3:I.Point_13)XIO(R2:4:O.Point_0)OTE(R2:2:O.Point_13);
   143: XIC(R2:3:I.Point_12)XIO(R2:2:O.Point_13)OTE(R2:2:O.Point_14);
   144: XIC(R2:3:I.Point_13)XIO(R2:2:O.Point_13)OTE(R2:2:O.Point_15);
   145: [XIC(R2:3:I.Point_14) XIO(R2:5:I.Point_0) ,XIC(R2:3:I.Point_15) XIC(R2:4:O.Point_0) XIO(R2:2:O.Point_14) XIO(R2:2:O.Point_15) ]XIO(B3[0].8)XIO(R2:4:O.Point_1)XIO(R2:2:O.Point_13)OTE(R2:4:O.Point_0);
